SUBAPPLICATION Uebung_125_sub (* Subapplication Type *)
  (* Standard: 61499-2 *)
  (* Version 1.0, 2025-10-22, franz *)
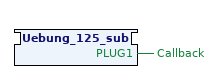
  PLUGS
    PLUG1 : isobus::pgn::tx::Callback;
  END_PLUGS
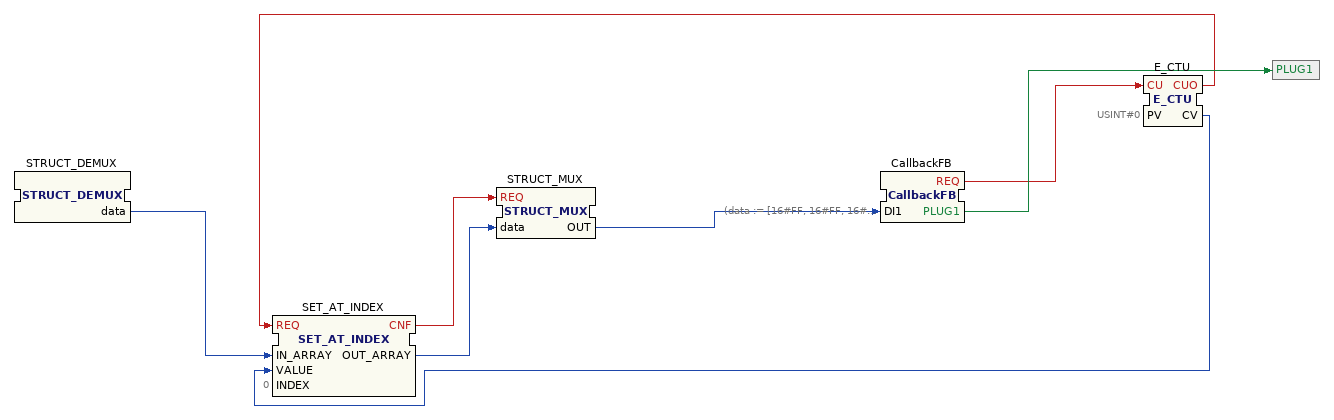
  FBS
    CallbackFB : isobus::pgn::tx::CallbackFB(DI1 := (data := [16#FF, 16#FF, 16#FF, 16#FF, 16#FF, 16#FF, 16#FF, 16#FF]));
    E_CTU : iec61499::events::E_CTU(PV := USINT#0);
    STRUCT_MUX : eclipse4diac::convert::STRUCT_MUX; {SET_ATTRIBUTE(StructuredType, isobus::pgn::CAN_MSG)}
    SET_AT_INDEX : eclipse4diac::utils::SET_AT_INDEX(INDEX := 0);
    STRUCT_DEMUX : eclipse4diac::convert::STRUCT_DEMUX; {SET_ATTRIBUTE(StructuredType, isobus::pgn::CAN_MSG)}
  END_FBS
  EVENT_CONNECTIONS
    CallbackFB.REQ TO E_CTU.CU;
    E_CTU.CUO TO SET_AT_INDEX.REQ;
    SET_AT_INDEX.CNF TO STRUCT_MUX.REQ;
  END_CONNECTIONS
  DATA_CONNECTIONS
    STRUCT_MUX.OUT TO CallbackFB.DI1;
    STRUCT_DEMUX.data TO SET_AT_INDEX.IN_ARRAY;
    E_CTU.CV TO SET_AT_INDEX.VALUE;
    SET_AT_INDEX.OUT_ARRAY TO STRUCT_MUX.data;
  END_CONNECTIONS
  ADAPTER_CONNECTIONS
    CallbackFB.PLUG1 TO PLUG1;
  END_CONNECTIONS
END_SUBAPPLICATION
